FUNCTION_BLOCK FB_SV_Logik
VAR_IN_OUT
	Steuerung	: ST_SV_Steuerung;
	Zustand		: ST_SV_Zustand;
END_VAR
VAR_INPUT
	Parameter	: ST_SV_Parameter;
END_VAR
VAR_OUTPUT
END_VAR
VAR
END_VAR

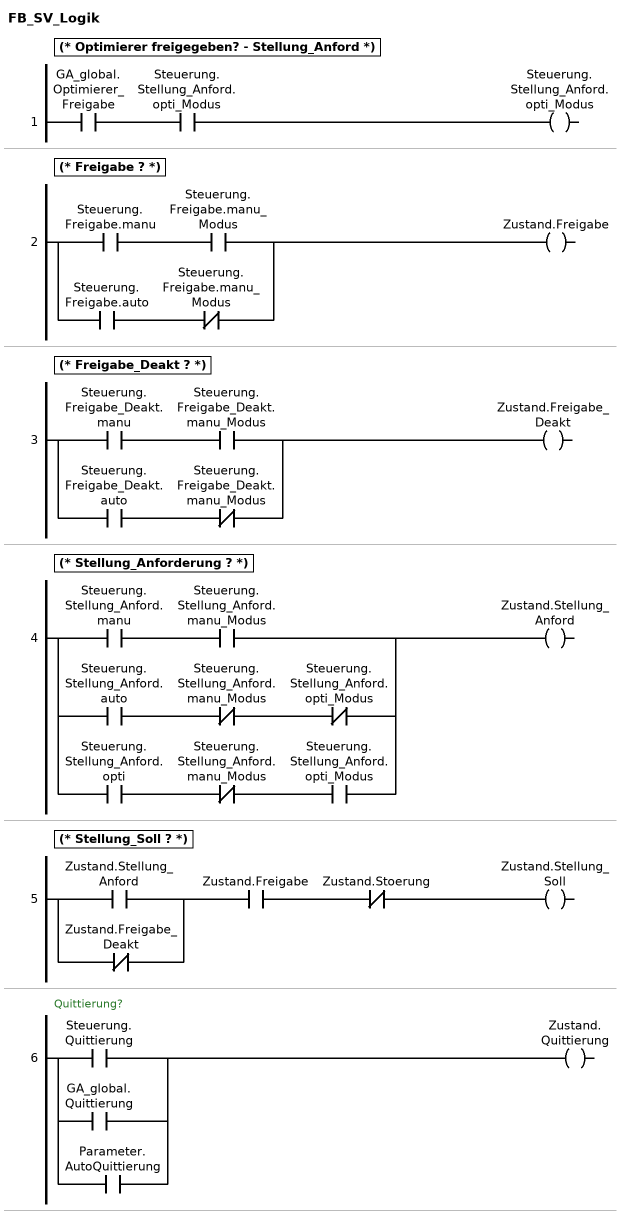
// NETWORK 1
// label: (* Optimierer freigegeben? - Stellung_Anford *)
Steuerung.Stellung_Anford.opti_Modus := GA_global.Optimierer_Freigabe AND Steuerung.Stellung_Anford.opti_Modus;

// NETWORK 2
// label: (* Freigabe ? *)
Zustand.Freigabe := Steuerung.Freigabe.manu AND Steuerung.Freigabe.manu_Modus OR Steuerung.Freigabe.auto AND NOT Steuerung.Freigabe.manu_Modus;

// NETWORK 3
// label: (* Freigabe_Deakt ? *)
Zustand.Freigabe_Deakt := Steuerung.Freigabe_Deakt.manu AND Steuerung.Freigabe_Deakt.manu_Modus OR Steuerung.Freigabe_Deakt.auto AND NOT Steuerung.Freigabe_Deakt.manu_Modus;

// NETWORK 4
// label: (* Stellung_Anforderung ? *)
Zustand.Stellung_Anford := Steuerung.Stellung_Anford.manu AND Steuerung.Stellung_Anford.manu_Modus OR Steuerung.Stellung_Anford.auto AND NOT Steuerung.Stellung_Anford.manu_Modus AND NOT Steuerung.Stellung_Anford.opti_Modus OR Steuerung.Stellung_Anford.opti AND NOT Steuerung.Stellung_Anford.manu_Modus AND Steuerung.Stellung_Anford.opti_Modus;

// NETWORK 5
// label: (* Stellung_Soll ? *)
Zustand.Stellung_Soll := (Zustand.Stellung_Anford OR NOT Zustand.Freigabe_Deakt) AND Zustand.Freigabe AND NOT Zustand.Stoerung;

// NETWORK 6
// Quittierung?
Zustand.Quittierung := Steuerung.Quittierung OR GA_global.Quittierung OR Parameter.AutoQuittierung;

END_FUNCTION_BLOCK

(* stored: Version 1.1.0.1, ProductVersion 3.1.4024.9
   POU FB_SV_Logik: Id {d4d84fa6-d7a9-4b39-9051-b931d5932f22}, SpecialFunc None *)
